Staubli VAL3: OpenFile.pgx

public program OpenFile(string x_sFile, bool& x_bRes)
begin
  //
  nFileHandle=$fileOpen(x_sFile,"w")
  if nFileHandle>=0 and nFileHandle<=9
    x_bRes=true
  else
    x_bRes=false
    logMsg("打开文件失败:"+x_sFile)
  endIf
end
